FUNCTION_BLOCK EL3602
VAR
	_io : EL36x2_Data;
	{attribute addProperty Name "WcState"}
	_wcState : WcStateInputToggle;
	{attribute addProperty Name "Info data"}
	_infoData : InfoDataAds;
END_VAR

PROPERTY IO : REFERENCE TO EL36x2_Data
GET
IO REF= _io;
END_GET
END_PROPERTY

PROPERTY WcState : REFERENCE TO WcStateInputToggle
GET
WcState REF= _wcState;
END_GET
END_PROPERTY

END_FUNCTION_BLOCK

(* stored: Version 1.1.0.1, ProductVersion 3.1.4024.9
   POU EL3602: Id {f156213d-aa9f-0cda-2b34-95f69acf11be}, SpecialFunc None
   Property IO: Id {9225f083-17ad-02c1-2640-0535f6ac1d1b}
   Get Get: Id {7a7a02a6-4138-00c5-1749-2dedc4c7fc26}
   Property WcState: Id {5a5e6d99-4f4f-0b70-22f2-dbe24c32e0d4}
   Get Get: Id {88719102-edab-0b5f-381a-aec463ea3e6c} *)
